TYPE ST_Machine_Sts :
	STRUCT
	END_STRUCT
END_TYPE

(* stored: Version 1.1.0.1
   DUT ST_Machine_Sts: Id {c25640e2-b92a-47ce-8a06-7f3d13e3f0d3} *)
